Staubli VAL3: robot2PLC.pgx

program robot2PLC()
  local num l_nLocalNum
  local num l_nNextNum
  local num l_ns
begin
  l_nLocalNum=-1
  while true
    //

    wait(dPlaceDone[0]==true or dPlaceDone[1]==true or dPlaceDone[2]==true or dPlaceDone[3]==true)
    //
    l_ns=clock()
    do
      delay(0)
    until clock()-l_ns>0.35

    if (dPlaceDone[0]==true)
      dPlaceDone[0]=false
    elseIf (dPlaceDone[1]==true)
      dPlaceDone[1]=false
    elseIf (dPlaceDone[2]==true)
      dPlaceDone[2]=false
    elseIf (dPlaceDone[3]==true)
      dPlaceDone[3]=false
    else
      dPlaceDone[0]=false
      dPlaceDone[1]=false
      dPlaceDone[2]=false
      dPlaceDone[3]=false
    endIf
    //
  endWhile
end
